FUNCTION_BLOCK FB_Lens_Test EXTENDS TcUnit.FB_TestSuite
VAR
    nTestID : INT;
    fbLens : FB_Lens;
END_VAR


nTestID := 0;


METHOD TestInvalidDeltaExpectError0FocalLength
VAR_INPUT
    fDelta : LREAL;
END_VAR

TEST(CONCAT('TestInvalidDeltaExpectError0FocalLength ID: ',
    INT_TO_STRING(nTestID))
);

fbCalcFocalLengthSingleLens(
    fDelta := fDelta,
    fRadius := 0.005,
    fFocalLength =>,
    bError =>,
    sErrorMsg =>
);

AssertTrue(
    Condition := fbCalcFocalLengthSingleLens.bError,
    Message := 'Expected bError bit to be true but it was false.'
);

AssertTrue(
    Condition := fbCalcFocalLengthSingleLens.sErrorMsg <> '',
    Message := 'Expected sErrorMsg to not be empty.'
);

AssertEquals_LREAL(
    Expected := 0,
    Actual := fbCalcFocalLengthSingleLens.fFocalLength,
    Delta := 0,
    Message := 'Calculated focal length should be 0 when an error is detected.'
);

TEST_FINISHED();

nTestID := nTestID + 1;
END_METHOD


METHOD TestValidInputsExpectNoErrorAccurateFocalLength
VAR_INPUT
    fDelta : LREAL;
    fRadius : LREAL;

    fExpected : LREAL;
END_VAR

TEST(CONCAT('TestValidInputsExpectNoErrorAccurateFocalLength ID: ',
    INT_TO_STRING(nTestID))
);

fbCalcFocalLengthSingleLens(
    fDelta := fDelta,
    fRadius := fRadius,
    fFocalLength =>,
    bError =>,
    sErrorMsg =>
);

AssertFalse(
    Condition := fbCalcFocalLengthSingleLens.bError,
    Message := 'Expected bError bit to be false but it was true.'
);

AssertFalse(
    Condition := fbCalcFocalLengthSingleLens.sErrorMsg <> '',
    Message := 'Expected sErrorMsg to be empty.'
);

AssertEquals_LREAL(
    Expected := fExpected,
    Actual := fbCalcFocalLengthSingleLens.fFocalLength,
    Delta := ABS(0.001 * fExpected),
    Message := 'Calculated focal length did not calculate close enough to the expected value.'
);

TEST_FINISHED();

nTestID := nTestID + 1;
END_METHOD

END_FUNCTION_BLOCK

(* stored: Version 1.1.0.1, ProductVersion 3.1.4022.18
   POU FB_Lens_Test: Id {9add33cb-e8c3-4b34-834a-827d76bb686e}, SpecialFunc None
   Method TestInvalidDeltaExpectError0FocalLength: Id {b8564aa5-bff1-429e-860c-b508ebb73485}
   Method TestValidInputsExpectNoErrorAccurateFocalLength: Id {f49502d8-148a-4213-9cbf-07c6f3490873} *)
